# EPICS substitutions: surfSafetyApp/Db/surf_safety.substitutions
file "$(TOP)/beckhoffApp/beckhoff_write_pv.template" {
    pattern {P, NAME, PORT, ADSPORT, V, RECTYPE, EPICSDTYP, ADS_TYPE}
    {"\$(P)", "ERROR_ACK:SP", "\$(PORT)", "\$(ADSPORT)", "GVL_SAFETY.ERROR_ACK", longout, "asynInt32", "BOOL"}
}

file "$(TOP)/beckhoffApp/beckhoff_read_pv.template" {
    pattern {P, NAME, PORT, ADSPORT, V, RECTYPE, EPICSDTYP, ADS_TYPE}
    {"\$(P)", "ERROR_ACK", "\$(PORT)", "\$(ADSPORT)", "GVL_SAFETY.ERROR_ACK", "longin", "asynInt32", "BOOL"}
}
